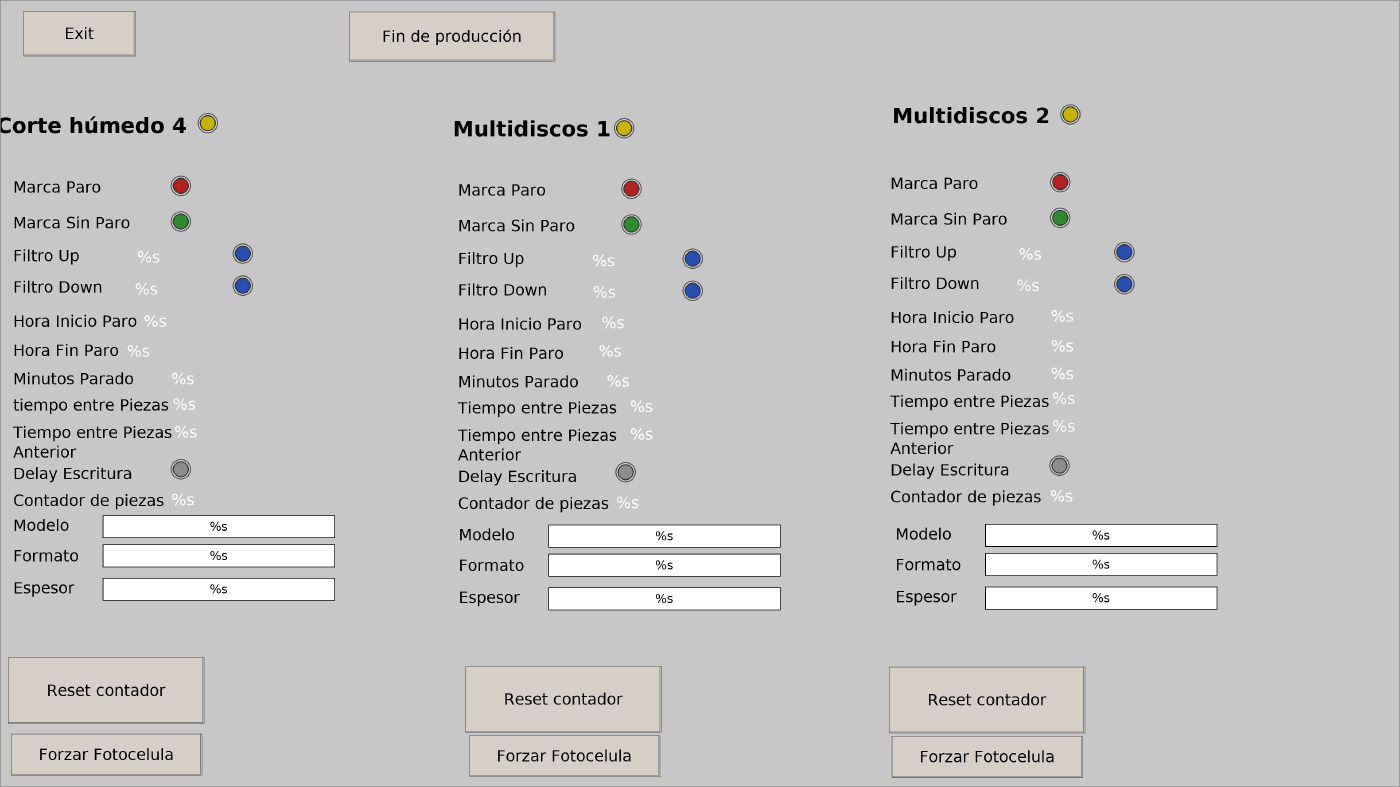
VISUALIZATION DiagnosticoFB  // 1920x1080
    Rectangle (185,338 93x30), "%s", text variable: FuncParoNodoCorteH4Remote1.Funci_CortHum4.tFiltro_up_Ftc.ET
    Label (10,146 231x53), "Corte húmedo 4"
    Label (15,242 150x30), "Marca Paro"
    Lamp1 (269,153 32x32), variable: FuncParoNodoCorteH4Remote1.Funci_CortHum4.Fotocelula, style: Lamp-Lamp1-Yellow
    Lamp1 (232,239 32x32), variable: FuncParoNodoCorteH4Remote1.Funci_CortHum4.MParo_Ftc, style: Lamp-Lamp1-Red
    Label (15,291 188x30), "Marca Sin Paro"
    Lamp1 (232,288 32x32), variable: FuncParoNodoCorteH4Remote1.Funci_CortHum4.M_SinParo_Ftc, style: Lamp-Lamp1-Green
    Label (15,336 117x30), "Filtro Up"
    Rectangle (182,382 93x30), "%s", text variable: FuncParoNodoCorteH4Remote1.Funci_CortHum4.tFiltro_down_Ftc.ET
    Label (15,379 143x30), "Filtro Down"
    Rectangle (194,426 183x30), "%s", text variable: FuncParoNodoCorteH4Remote1.Funci_CortHum4.H_InParo_Ftc
    Label (15,426 204x30), "Hora Inicio Paro"
    Lamp1 (317,332 32x32), variable: FuncParoNodoCorteH4Remote1.Funci_CortHum4.tFiltro_up_Ftc.Q, style: Lamp-Lamp1-Blue
    Lamp1 (317,376 32x32), variable: FuncParoNodoCorteH4Remote1.Funci_CortHum4.tFiltro_down_Ftc.Q, style: Lamp-Lamp1-Blue
    Rectangle (171,467 179x30), "%s", text variable: FuncParoNodoCorteH4Remote1.Funci_CortHum4.H_FinParo_Ftc
    Label (15,466 204x30), "Hora Fin Paro"
    Rectangle (232,505 192x30), "%s", text variable: FuncParoNodoCorteH4Remote1.Funci_CortHum4.Min_Parado_Ftc
    Label (15,505 204x30), "Minutos Parado"
    Label (15,541 244x30), "tiempo entre Piezas"
    Label (15,576 255x62), "Tiempo entre Piezas Anterior"
    Label (15,635 204x30), "Delay Escritura"
    Rectangle (232,671 93x30), "%s", text variable: FuncParoNodoCorteH4Remote1.Funci_CortHum4.Cont_Piezas_Ftc
    Label (15,672 215x30), "Contador de piezas"
    Lamp1 (232,628 32x32), variable: FuncParoNodoCorteH4Remote1.Funci_CortHum4.Delay_Esc_Ftc.Q, style: Lamp-Lamp1-Gray
    Button (32,15 154x62), "Exit"
        OnMouseClick: change screen: Home_CortH4
    Rectangle (809,343 93x30), "%s", text variable: FuncParoNodoMultidiscos.Funci_Multidiscos1.tFiltro_up_Ftc.ET
    Label (614,134 231x86), "Multidiscos 1"
    Label (625,246 150x30), "Marca Paro"
    Lamp1 (840,160 32x32), variable: FuncParoNodoMultidiscos.Funci_Multidiscos1.Fotocelula, style: Lamp-Lamp1-Yellow
    Lamp1 (850,243 32x32), variable: FuncParoNodoMultidiscos.Funci_Multidiscos1.MParo_Ftc, style: Lamp-Lamp1-Red
    Label (625,295 188x30), "Marca Sin Paro"
    Lamp1 (850,292 32x32), variable: FuncParoNodoMultidiscos.Funci_Multidiscos1.M_SinParo_Ftc, style: Lamp-Lamp1-Green
    Label (625,340 117x30), "Filtro Up"
    Rectangle (810,386 93x30), "%s", text variable: FuncParoNodoMultidiscos.Funci_Multidiscos1.tFiltro_down_Ftc.ET
    Label (625,383 143x30), "Filtro Down"
    Rectangle (822,428 183x30), "%s", text variable: FuncParoNodoMultidiscos.Funci_Multidiscos1.H_InParo_Ftc
    Label (625,430 204x30), "Hora Inicio Paro"
    Lamp1 (934,339 32x32), variable: FuncParoNodoMultidiscos.Funci_Multidiscos1.tFiltro_up_Ftc.Q, style: Lamp-Lamp1-Blue
    Lamp1 (934,383 32x32), variable: FuncParoNodoMultidiscos.Funci_Multidiscos1.tFiltro_down_Ftc.Q, style: Lamp-Lamp1-Blue
    Rectangle (818,467 179x30), "%s", text variable: FuncParoNodoMultidiscos.Funci_Multidiscos1.H_FinParo_Ftc
    Label (625,470 204x30), "Hora Fin Paro"
    Rectangle (829,508 192x30), "%s", text variable: FuncParoNodoMultidiscos.Funci_Multidiscos1.Min_Parado_Ftc
    Label (625,509 204x30), "Minutos Parado"
    Label (625,545 244x30), "Tiempo entre Piezas"
    Label (625,580 255x62), "Tiempo entre Piezas Anterior"
    Label (625,639 204x30), "Delay Escritura"
    Rectangle (842,675 93x30), "%s", text variable: FuncParoNodoMultidiscos.Funci_Multidiscos1.Cont_Piezas_Ftc
    Label (625,676 215x30), "Contador de piezas"
    Lamp1 (842,632 32x32), variable: FuncParoNodoMultidiscos.Funci_Multidiscos1.Delay_Esc_Ftc.Q, style: Lamp-Lamp1-Gray
    Rectangle (1394,334 93x30), "%s", text variable: FuncParoNodoMultidiscos.Funci_Multidiscos2.tFiltro_up_Ftc.ET
    Label (1207,115 250x88), "Multidiscos 2"
    Label (1218,237 150x30), "Marca Paro"
    Lamp1 (1452,141 32x32), variable: FuncParoNodoMultidiscos.Funci_Multidiscos2.Fotocelula, style: Lamp-Lamp1-Yellow
    Lamp1 (1438,234 32x32), variable: FuncParoNodoMultidiscos.Funci_Multidiscos2.MParo_Ftc, style: Lamp-Lamp1-Red
    Label (1218,286 188x30), "Marca Sin Paro"
    Lamp1 (1438,283 32x32), variable: FuncParoNodoMultidiscos.Funci_Multidiscos2.M_SinParo_Ftc, style: Lamp-Lamp1-Green
    Label (1218,331 117x30), "Filtro Up"
    Rectangle (1391,377 93x30), "%s", text variable: FuncParoNodoMultidiscos.Funci_Multidiscos2.tFiltro_down_Ftc.ET
    Label (1218,374 143x30), "Filtro Down"
    Rectangle (1438,419 183x30), "%s", text variable: FuncParoNodoMultidiscos.Funci_Multidiscos2.H_InParo_Ftc
    Label (1218,421 204x30), "Hora Inicio Paro"
    Lamp1 (1526,330 32x32), variable: FuncParoNodoMultidiscos.Funci_Multidiscos2.tFiltro_up_Ftc.Q, style: Lamp-Lamp1-Blue
    Lamp1 (1526,374 32x32), variable: FuncParoNodoMultidiscos.Funci_Multidiscos2.tFiltro_down_Ftc.Q, style: Lamp-Lamp1-Blue
    Rectangle (1438,460 179x30), "%s", text variable: FuncParoNodoMultidiscos.Funci_Multidiscos2.H_FinParo_Ftc
    Label (1218,461 204x30), "Hora Fin Paro"
    Rectangle (1438,498 192x30), "%s", text variable: FuncParoNodoMultidiscos.Funci_Multidiscos2.Min_Parado_Ftc
    Label (1218,500 204x30), "Minutos Parado"
    Label (1218,536 244x30), "Tiempo entre Piezas"
    Label (1218,571 255x62), "Tiempo entre Piezas Anterior"
    Label (1218,630 204x30), "Delay Escritura"
    Rectangle (1437,666 93x30), "%s", text variable: FuncParoNodoMultidiscos.Funci_Multidiscos2.Cont_Piezas_Ftc
    Label (1218,667 215x30), "Contador de piezas"
    Lamp1 (1437,623 32x32), variable: FuncParoNodoMultidiscos.Funci_Multidiscos2.Delay_Esc_Ftc.Q, style: Lamp-Lamp1-Gray
    Rectangle (234,540 192x30), "%s", text variable: FuncParoNodoCorteH4Remote1.Funci_CortHum4.t_Entre_Piez_Ftc
    Rectangle (861,543 192x30), "%s", text variable: FuncParoNodoMultidiscos.Funci_Multidiscos1.t_Entre_Piez_Ftc
    Rectangle (1440,532 192x30), "%s", text variable: FuncParoNodoMultidiscos.Funci_Multidiscos2.t_Entre_Piez_Ftc
    Rectangle (236,578 192x30), "%s", text variable: FuncParoNodoCorteH4Remote1.Funci_CortHum4.t_Entr_Piez_Ante_Ftc
    Rectangle (861,581 192x30), "%s", text variable: FuncParoNodoMultidiscos.Funci_Multidiscos1.t_Entr_Piez_Ante_Ftc
    Rectangle (1440,570 192x30), "%s", text variable: FuncParoNodoMultidiscos.Funci_Multidiscos2.t_Entr_Piez_Ante_Ftc
    Button (11,902 269x91), "Reset contador"
        tap FuncParoNodoCorteH4Remote1.Funci_CortHum4.ResetContPiez
    Button (638,914 269x91), "Reset contador"
        tap FuncParoNodoMultidiscos.Funci_Multidiscos1.ResetContPiez
    Button (1219,915 269x91), "Reset contador"
        tap FuncParoNodoMultidiscos.Funci_Multidiscos2.ResetContPiez
    Button (643,1009 262x57), "Forzar Fotocelula"
        tap FuncParoNodoMultidiscos.ForzadoFtcMultidiscos1
    Button (1223,1010 262x57), "Forzar Fotocelula"
        tap FuncParoNodoMultidiscos.ForzadoFtc2_Multidiscos2
    Button (15,1007 262x57), "Forzar Fotocelula"
        tap FuncParoNodoCorteH4Remote1.ForzadoFtcCortHum4
    Button (479,16 282x68), "Fin de producción"
        OnMouseClick: OpenDialog Dialog=V_Emerg_Fin_Prod_Ch4, OpenModal=True, OpenCentered=True
    Label (15,706 92x30), "Modelo"
    Label (15,748 105x30), "Formato"
    Label (15,792 99x30), "Espesor"
    Rectangle (141,707 318x31), "%s", text variable: FuncParoNodoCorteH4Remote1.FunGeneCortHum4.s_ModeloActualTabla
        OnMouseDown: write the text variable via Edit
    Rectangle (141,747 318x31), "%s", text variable: FuncParoNodoCorteH4Remote1.FunGeneCortHum4.s_FormatoActualTabla
        OnMouseDown: write the text variable via Edit
    Rectangle (141,793 318x31), "%s", text variable: FuncParoNodoCorteH4Remote1.FunGeneCortHum4.s_EspesorActualTabla
        OnMouseDown: write the text variable via Edit
    Label (626,719 92x30), "Modelo"
    Label (626,761 105x30), "Formato"
    Label (626,805 99x30), "Espesor"
    Rectangle (752,720 318x31), "%s", text variable: FuncParoNodoMultidiscos.FunGeneMultidiscos1.s_ModeloActualTabla
        OnMouseDown: write the text variable via Edit
    Rectangle (752,760 318x31), "%s", text variable: FuncParoNodoMultidiscos.FunGeneMultidiscos1.s_FormatoActualTabla
        OnMouseDown: write the text variable via Edit
    Rectangle (752,806 318x31), "%s", text variable: FuncParoNodoMultidiscos.FunGeneMultidiscos1.s_EspesorActualTabla
        OnMouseDown: write the text variable via Edit
    Label (1225,718 92x30), "Modelo"
    Label (1225,760 105x30), "Formato"
    Label (1225,804 99x30), "Espesor"
    Rectangle (1351,719 318x31), "%s", text variable: FuncParoNodoMultidiscos.FunGeneMultidiscos2.s_ModeloActualTabla
        OnMouseDown: write the text variable via Edit
    Rectangle (1351,759 318x31), "%s", text variable: FuncParoNodoMultidiscos.FunGeneMultidiscos2.s_FormatoActualTabla
        OnMouseDown: write the text variable via Edit
    Rectangle (1351,805 318x31), "%s", text variable: FuncParoNodoMultidiscos.FunGeneMultidiscos2.s_EspesorActualTabla
        OnMouseDown: write the text variable via Edit
END_VISUALIZATION

(* stored: Version 1.1.0.1, ProductVersion 3.1.4024.12
   Visu DiagnosticoFB: Id {0e784541-fdbe-4048-8d88-3d9ad672f9bb} *)
